// TIA Portal V16 export
// export: Created 2022-11-17T15:49:38.8792382Z, ExportSetting WithDefaults, DisplayName Totally Integrated Automation Portal, DisplayVersion V16 Update 6, DisplayName TIA Portal Version Control Interface, DisplayVersion V16 Update 2, DisplayName TIA Portal Openness, DisplayVersion V16 Update 6, DisplayName SINAMICS Startdrive Advanced, DisplayVersion V16 Update 5, DisplayName SINAMICS Startdrive G130, G150, S120, S150, SINAMICS MV, S210, DisplayVersion V16 Update 5, DisplayName SINAMICS Startdrive G110M, G120, G120C, G120D, G120P, G115D, DisplayVersion V16 Update 5, DisplayName STEP 7 Professional, DisplayVersion V16 Update 6, DisplayName STEP 7 Safety, DisplayVersion V16, DisplayName WinCC Advanced, DisplayVersion V16 Update 6
DATA_BLOCK "DB18_TableSpeed"   // DB18
{ S7_Optimized_Access := 'FALSE' }
VERSION : 0.1
// stored: AutoNumber false, IsOnlyStoredInLoadMemory false, IsWriteProtectedInAS false
   VAR RETAIN
      spare0 : Int := 0;
      spare1 : Int := 0;
      spare2 : Int := 0;
      spare3 : Int := 0;
      spare4 : Int := 0;
      spare5 : Int := 0;
      spare6 : Int := 0;
      spare7 : Int := 0;
      DBD16 : Real := 0.0;   // Actual speed in degrees per second (split before use)
      DBD20 : Real := 90.0;   // Low speed in degrees per second (split before use)
      DBD24 : Real := 900.0;   // High speed in degrees per second (split before use)
      spare14 : Int := 0;
      DBW30 : Int := 0;   // Degrees to reach minimum speed from maximum speed
      spare16 : Int := 0;
      DBW34 : Int := 50;
   END_VAR
BEGIN
END_DATA_BLOCK
